// Mitsubishi GX Works2 project: Conveyor2   PLC: Q02U

PROGRAM MAIN
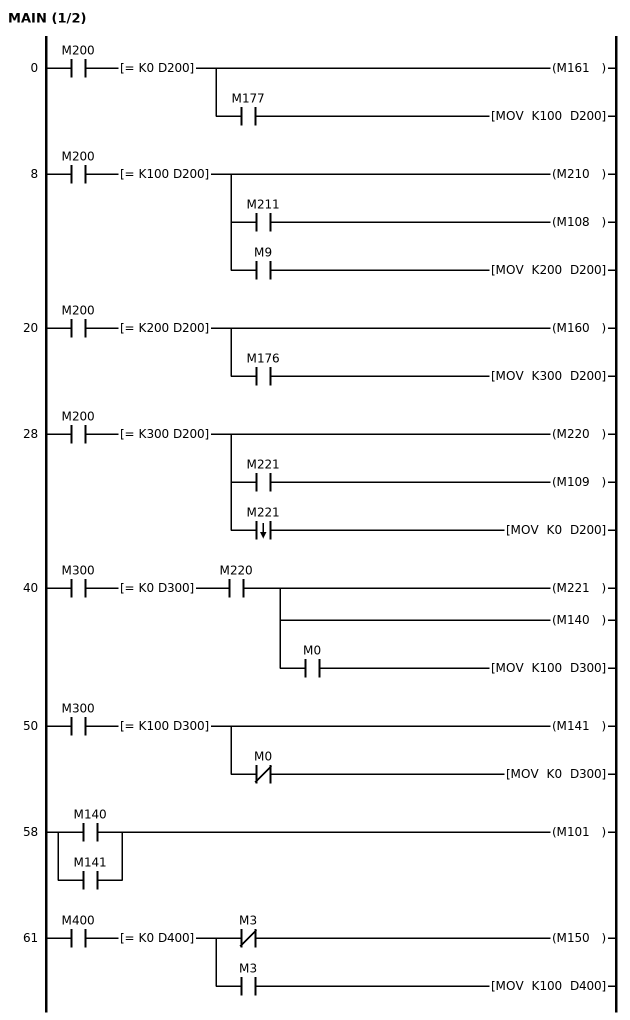
0     LD      M200
      AND=    K0 D200
      OUT     M161
      AND     M177
      MOV     K100 D200
8     LD      M200
      AND=    K100 D200
      OUT     M210
      MPS
      AND     M211
      OUT     M108
      MPP
      AND     M9
      MOV     K200 D200
20    LD      M200
      AND=    K200 D200
      OUT     M160
      AND     M176
      MOV     K300 D200
28    LD      M200
      AND=    K300 D200
      OUT     M220
      MPS
      AND     M221
      OUT     M109
      MPP
      ANDF    M221
      MOV     K0 D200
40    LD      M300
      AND=    K0 D300
      AND     M220
      OUT     M221
      OUT     M140
      AND     M0
      MOV     K100 D300
50    LD      M300
      AND=    K100 D300
      OUT     M141
      ANI     M0
      MOV     K0 D300
58    LD      M140
      OR      M141
      OUT     M101
61    LD      M400
      AND=    K0 D400
      MPS
      ANI     M3
      OUT     M150
      MPP
      AND     M3
      MOV     K100 D400
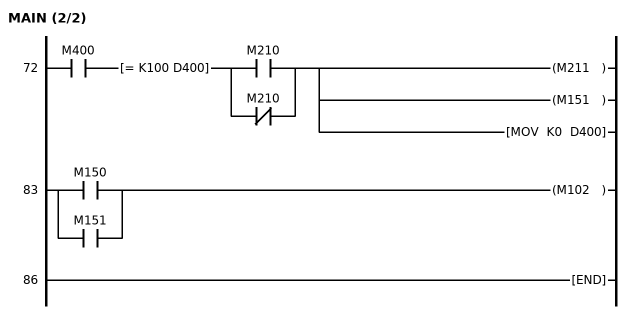
72    LD      M400
      AND=    K100 D400
      LD      M210
      ORI     M210
      ANB
      OUT     M211
      OUT     M151
      MOV     K0 D400
83    LD      M150
      OR      M151
      OUT     M102
86    END
END_PROGRAM

PROGRAM INPUT
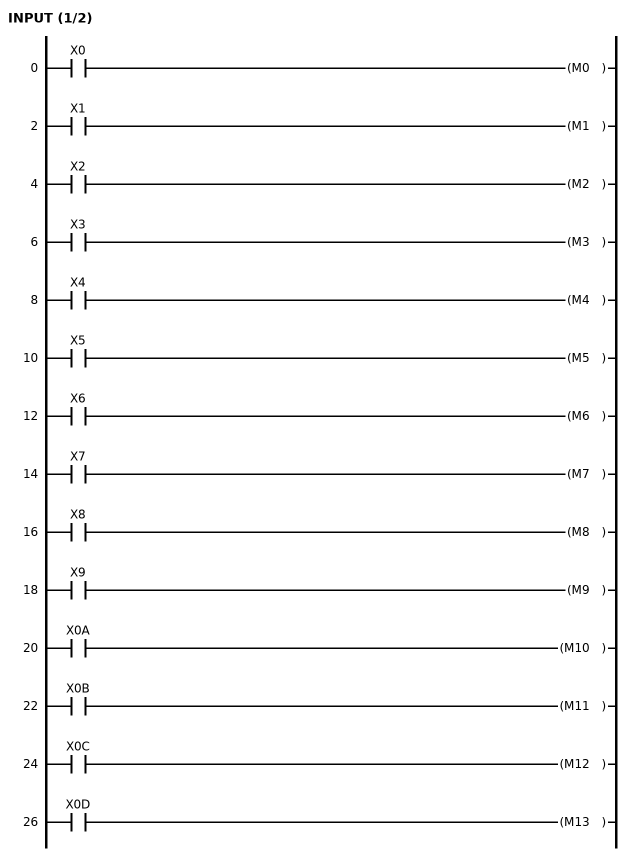
0     LD      X0
      OUT     M0
2     LD      X1
      OUT     M1
4     LD      X2
      OUT     M2
6     LD      X3
      OUT     M3
8     LD      X4
      OUT     M4
10    LD      X5
      OUT     M5
12    LD      X6
      OUT     M6
14    LD      X7
      OUT     M7
16    LD      X8
      OUT     M8
18    LD      X9
      OUT     M9
20    LD      X0A
      OUT     M10
22    LD      X0B
      OUT     M11
24    LD      X0C
      OUT     M12
26    LD      X0D
      OUT     M13
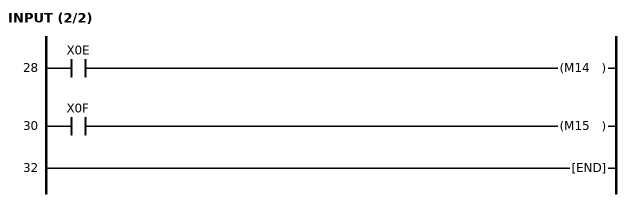
28    LD      X0E
      OUT     M14
30    LD      X0F
      OUT     M15
32    END
END_PROGRAM

PROGRAM OUTPUT
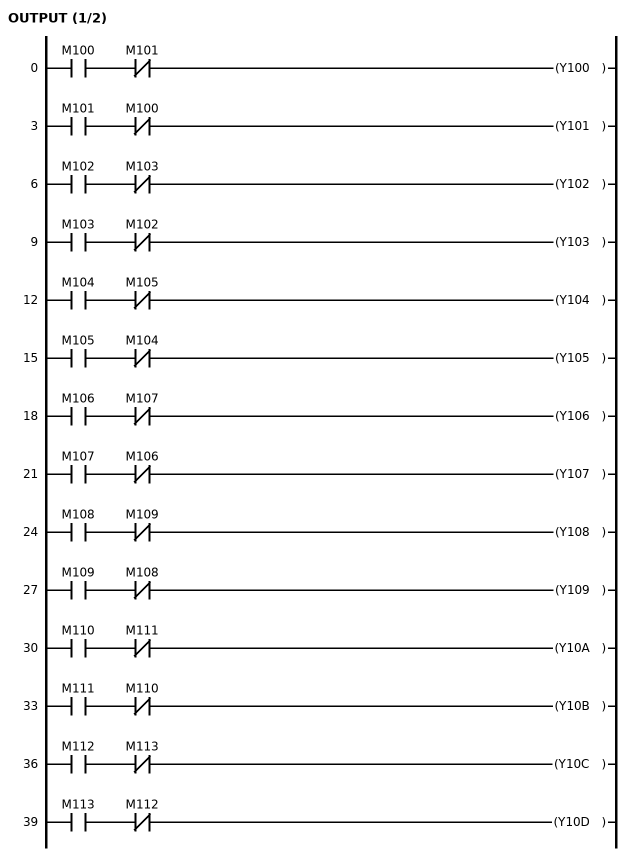
0     LD      M100
      ANI     M101
      OUT     Y100
3     LD      M101
      ANI     M100
      OUT     Y101
6     LD      M102
      ANI     M103
      OUT     Y102
9     LD      M103
      ANI     M102
      OUT     Y103
12    LD      M104
      ANI     M105
      OUT     Y104
15    LD      M105
      ANI     M104
      OUT     Y105
18    LD      M106
      ANI     M107
      OUT     Y106
21    LD      M107
      ANI     M106
      OUT     Y107
24    LD      M108
      ANI     M109
      OUT     Y108
27    LD      M109
      ANI     M108
      OUT     Y109
30    LD      M110
      ANI     M111
      OUT     Y10A
33    LD      M111
      ANI     M110
      OUT     Y10B
36    LD      M112
      ANI     M113
      OUT     Y10C
39    LD      M113
      ANI     M112
      OUT     Y10D
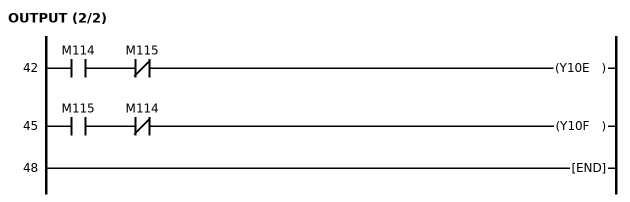
42    LD      M114
      ANI     M115
      OUT     Y10E
45    LD      M115
      ANI     M114
      OUT     Y10F
48    END
END_PROGRAM
